(* IEC 61131-3 sources: inproshop/TEAM_V2.0-demo_exported/OP80/1.Global, 7 files *)

(* ---- DB8000_Control.st ---- *)
VAR_GLOBAL
	Mode:Str_Mode;
	HMI:Str_HMI;
END_VAR
VAR_GLOBAL RETAIN PERSISTENT
	Machine AT %MB131496 : Str_Machine;
END_VAR

(* ---- DB8002_Recipe.st ---- *)
VAR_GLOBAL
END_VAR
VAR_GLOBAL RETAIN PERSISTENT

	RecipeChangePmt AT %MB131099 : BOOL;	//配方允许切换
	ParameterChangePmt AT %MB131224 : BOOL;	//参数允许更改
	RecipeNumTemp AT %MB131225 : INT;	//HMI选中还未保存到PLC的编号.
	RecipeNum AT %MB131227 : INT;	//配方元素编号.
	RecipeName AT %MB131576 : STRING(20);	//配方元素名称.
	RecipeNameTemp AT %MB131597 : STRING(20);	//HMI头部显示当前配方名称
	RecipeOk AT %MB131229 : BOOL;//配方可用
	DownLoad AT %MB131230 : BOOL;//配方下载
	TypeDataCur AT %MB131620 : Str_OP80_Recipe;//当前配方
	TypeData AT %MB131648 : ARRAY [0..20] OF Str_OP80_Recipe;//配方数据
END_VAR

(* ---- DB8003_Count.st ---- *)
VAR_GLOBAL RETAIN PERSISTENT
	Total AT %MB238216 : Str_Count;//总计数
	OK AT %MB238888 : Str_Count;//OK计数
	NG AT %MB239560 : Str_Count;//NG计数
END_VAR
VAR_GLOBAL
	Yield : REAL;//良品率
	Clear : BOOL;//清除计数
END_VAR

(* ---- DB8005_Communication.st ---- *)
VAR_GLOBAL
	TcpClient:ARRAY[0..9] OF Str_TcpClient;
	TcpSever:ARRAY[0..9] OF Str_TcpClient;
	From_OPXX    :Str_OP80_TO_OPXX;
	TO_OPXX    :Str_OPXX_TO_OP80;
	FromMaster  :Str_FromMaster;
END_VAR

(* ---- DB8050_DriveControl.st ---- *)
VAR_GLOBAL RETAIN PERSISTENT
	CylCtrl AT %MB133808 : ARRAY [0..63] OF Str_Cylinder;
	VacCtrl AT %MB146812 : ARRAY [0..63] OF Str_Cylinder;
	AxisCtrl AT %MB179816 : ARRAY [0..16] OF Str_Axis;
	Sensor AT %MB155388 : ARRAY [0..168] OF Str_Sensor;
	CamCtrl AT %MB131084 : ARRAY [1..3] OF Str_CamControl;
	HeatCtrl AT %MB131100 : ARRAY [1..1] OF Str_Heating;
	AgingCtrl AT %MB209056 : ARRAY [0..80] OF Str_Aging;
	AirLeakCtrl AT %MB131268 : ARRAY [0..2] OF Str_AirLeak;
	PalletCtrl AT %MB131144 : ARRAY [0..3] OF Str_Palletizing;
END_VAR

VAR_GLOBAL
	DoubleStart:ARRAY [1..4] OF Str_DoubleStart;
	Epson : ARRAY [1..10] OF Str_Epson;
	Kuka : ARRAY [1..2] OF Str_Kuka6;
	Rotdisk:ARRAY [1..1] OF Str_Rotdisk;
	Stopper:ARRAY [1..20] OF Str_Stopper;
	Motor:ARRAY [1..10] OF Str_Motor;
	AI:ARRAY [0..200] OF Str_AI;
	GearCtrl:ARRAY [1..1] OF Str_Gear;
	AAS:ARRAY [1..1] OF Str_AAS;
END_VAR

(* ---- DB8070_Fault.st ---- *)
VAR_GLOBAL
	Estop:Str_OP80_FaultEstop;//紧急停止类报警
	Stop:Str_OP80_Faultstop;//暂停类报警
	Run:Str_OP80_FaultRun;//警告类报警
	EstopTotal:BOOL;//急停报警汇总
	StopTotal:BOOL;//暂停报警汇总
	RunTotal:BOOL;//警告汇总
END_VAR

(* ---- DB8090_Other.st ---- *)
VAR_GLOBAL RETAIN PERSISTENT
	{attribute 'ElemComment':='(),(上料机械臂取料夹爪),(上料机械臂放料夹爪),(缓存台1),(缓存台2),(缓存台3),(缓存台4),(测试台1),(测试台2),(测试台3),(测试台4),(下料机械臂),4()'}
	StationData AT %MB142384 : ARRAY [0..15] OF Str_OP80_StationData;
	AgingTime AT %MB131231 : INT;//老化时间
	AgingInterval AT %MB131233 : INT;//老化间隔
	Product AT %MB220072 : ARRAY [0..20] OF Str_OP80_Product;
	Cyl_B_Sport AT %MB131235 : BOOL;//封堵B气缸是否动作

END_VAR
